// TIA Portal V16 export
// export: Created 2021-11-12T13:31:14.5106173Z, ExportSetting WithDefaults, DisplayName Totally Integrated Automation Portal, DisplayVersion V16 Update 3, DisplayName TIA Portal Version Control Interface, DisplayVersion V16 Update 2, DisplayName TIA Portal Openness, DisplayVersion V16 Update 3, DisplayName SINAMICS Startdrive Advanced, DisplayVersion V16 Update 5, DisplayName SINAMICS Startdrive G130, G150, S120, S150, SINAMICS MV, S210, DisplayVersion V16 Update 5, DisplayName SINAMICS Startdrive G110M, G120, G120C, G120D, G120P, G115D, DisplayVersion V16 Update 5, DisplayName STEP 7 Professional, DisplayVersion V16 Update 3, DisplayName STEP 7 Safety, DisplayVersion V16, DisplayName WinCC UA Professional, DisplayVersion V16 Update 3
FUNCTION_BLOCK "STD_RobotZones"   // FB39, LAD
{ S7_Optimized_Access := 'TRUE' }
VERSION : 0.1
// stored: AutoNumber true, IsIECCheckEnabled false, IsRetainMemResEnabled false, MemoryReserve 100, SetENOAutomatically false, UDAEnableTagReadback false
   VAR_INPUT
      IS_Rob1_ZoneRel : Struct
         Request : Bool;   // Robot requests entering the Station
         Rel : Bool;   // Robot is out of station area
      END_STRUCT;
      IS_Rob2_ZoneRel : Struct
         Request : Bool;   // Robot requests entering the Station
         Rel : Bool;   // Robot is out of station area
      END_STRUCT;
      IS_Rob3_ZoneRel : Struct
         Request : Bool;   // Robot requests entering the Station
         Rel : Bool;   // Robot is out of station area
      END_STRUCT;
      IS_Rob4_ZoneRel : Struct
         Request : Bool;   // Robot requests entering the Station
         Rel : Bool;   // Robot is out of station area
      END_STRUCT;
      IS_Rob5_ZoneRel : Struct
         Request : Bool;   // Robot requests entering the Station
         Rel : Bool;   // Robot is out of station area
      END_STRUCT;
      IS_Rob6_ZoneRel : Struct
         Request : Bool;   // Robot requests entering the Station
         Rel : Bool;   // Robot is out of station area
      END_STRUCT;
      IS_Rob7_ZoneRel : Struct
         Request : Bool;   // Robot requests entering the Station
         Rel : Bool;   // Robot is out of station area
      END_STRUCT;
      IS_Rob8_ZoneRel : Struct
         Request : Bool;   // Robot requests entering the Station
         Rel : Bool;   // Robot is out of station area
      END_STRUCT;
      IB1ZoneRelease : Bool;
   END_VAR
   VAR_OUTPUT
      OS_Rob1_ZoneAll : Struct
         Allowed : Bool;   // Station is allowed for robot entering
      END_STRUCT;
      OS_Rob2_ZoneAll : Struct
         Allowed : Bool;   // Station is allowed for robot entering
      END_STRUCT;
      OS_Rob3_ZoneAll : Struct
         Allowed : Bool;   // Station is allowed for robot entering
      END_STRUCT;
      OS_Rob4_ZoneAll : Struct
         Allowed : Bool;   // Station is allowed for robot entering
      END_STRUCT;
      OS_Rob5_ZoneAll : Struct
         Allowed : Bool;   // Station is allowed for robot entering
      END_STRUCT;
      OS_Rob6_ZoneAll : Struct
         Allowed : Bool;   // Station is allowed for robot entering
      END_STRUCT;
      OS_Rob7_ZoneAll : Struct
         Allowed : Bool;   // Station is allowed for robot entering
      END_STRUCT;
      OS_Rob8_ZoneAll : Struct
         Allowed : Bool;   // Station is allowed for robot entering
      END_STRUCT;
   END_VAR
   VAR_TEMP
      "TB1Zone free" : Bool;
      TS_Rob1_ZoneRel : Struct
         Request : Bool;   // Robot requests entering the Station
         Rel : Bool;   // Robot is out of station area
      END_STRUCT;
      TS_Rob2_ZoneRel : Struct
         Request : Bool;   // Robot requests entering the Station
         Rel : Bool;   // Robot is out of station area
      END_STRUCT;
      TS_Rob3_ZoneRel : Struct
         Request : Bool;   // Robot requests entering the Station
         Rel : Bool;   // Robot is out of station area
      END_STRUCT;
      TS_Rob4_ZoneRel : Struct
         Request : Bool;   // Robot requests entering the Station
         Rel : Bool;   // Robot is out of station area
      END_STRUCT;
      TS_Rob5_ZoneRel : Struct
         Request : Bool;   // Robot requests entering the Station
         Rel : Bool;   // Robot is out of station area
      END_STRUCT;
      TS_Rob6_ZoneRel : Struct
         Request : Bool;   // Robot requests entering the Station
         Rel : Bool;   // Robot is out of station area
      END_STRUCT;
      TS_Rob7_ZoneRel : Struct
         Request : Bool;   // Robot requests entering the Station
         Rel : Bool;   // Robot is out of station area
      END_STRUCT;
      TS_Rob8_ZoneRel : Struct
         Request : Bool;   // Robot requests entering the Station
         Rel : Bool;   // Robot is out of station area
      END_STRUCT;
      TS_Rob1_ZoneAll : Struct
         Allowed : Bool;   // Station is allowed for robot entering
      END_STRUCT;
      TS_Rob2_ZoneAll : Struct
         Allowed : Bool;   // Station is allowed for robot entering
      END_STRUCT;
      TS_Rob3_ZoneAll : Struct
         Allowed : Bool;   // Station is allowed for robot entering
      END_STRUCT;
      TS_Rob4_ZoneAll : Struct
         Allowed : Bool;   // Station is allowed for robot entering
      END_STRUCT;
      TS_Rob5_ZoneAll : Struct
         Allowed : Bool;   // Station is allowed for robot entering
      END_STRUCT;
      TS_Rob6_ZoneAll : Struct
         Allowed : Bool;   // Station is allowed for robot entering
      END_STRUCT;
      TS_Rob7_ZoneAll : Struct
         Allowed : Bool;   // Station is allowed for robot entering
      END_STRUCT;
      TS_Rob8_ZoneAll : Struct
         Allowed : Bool;   // Station is allowed for robot entering
      END_STRUCT;
      TB1ZoneRelease : Bool;
   END_VAR
BEGIN

REGION Network 1: *************** Clear Temporary ***************
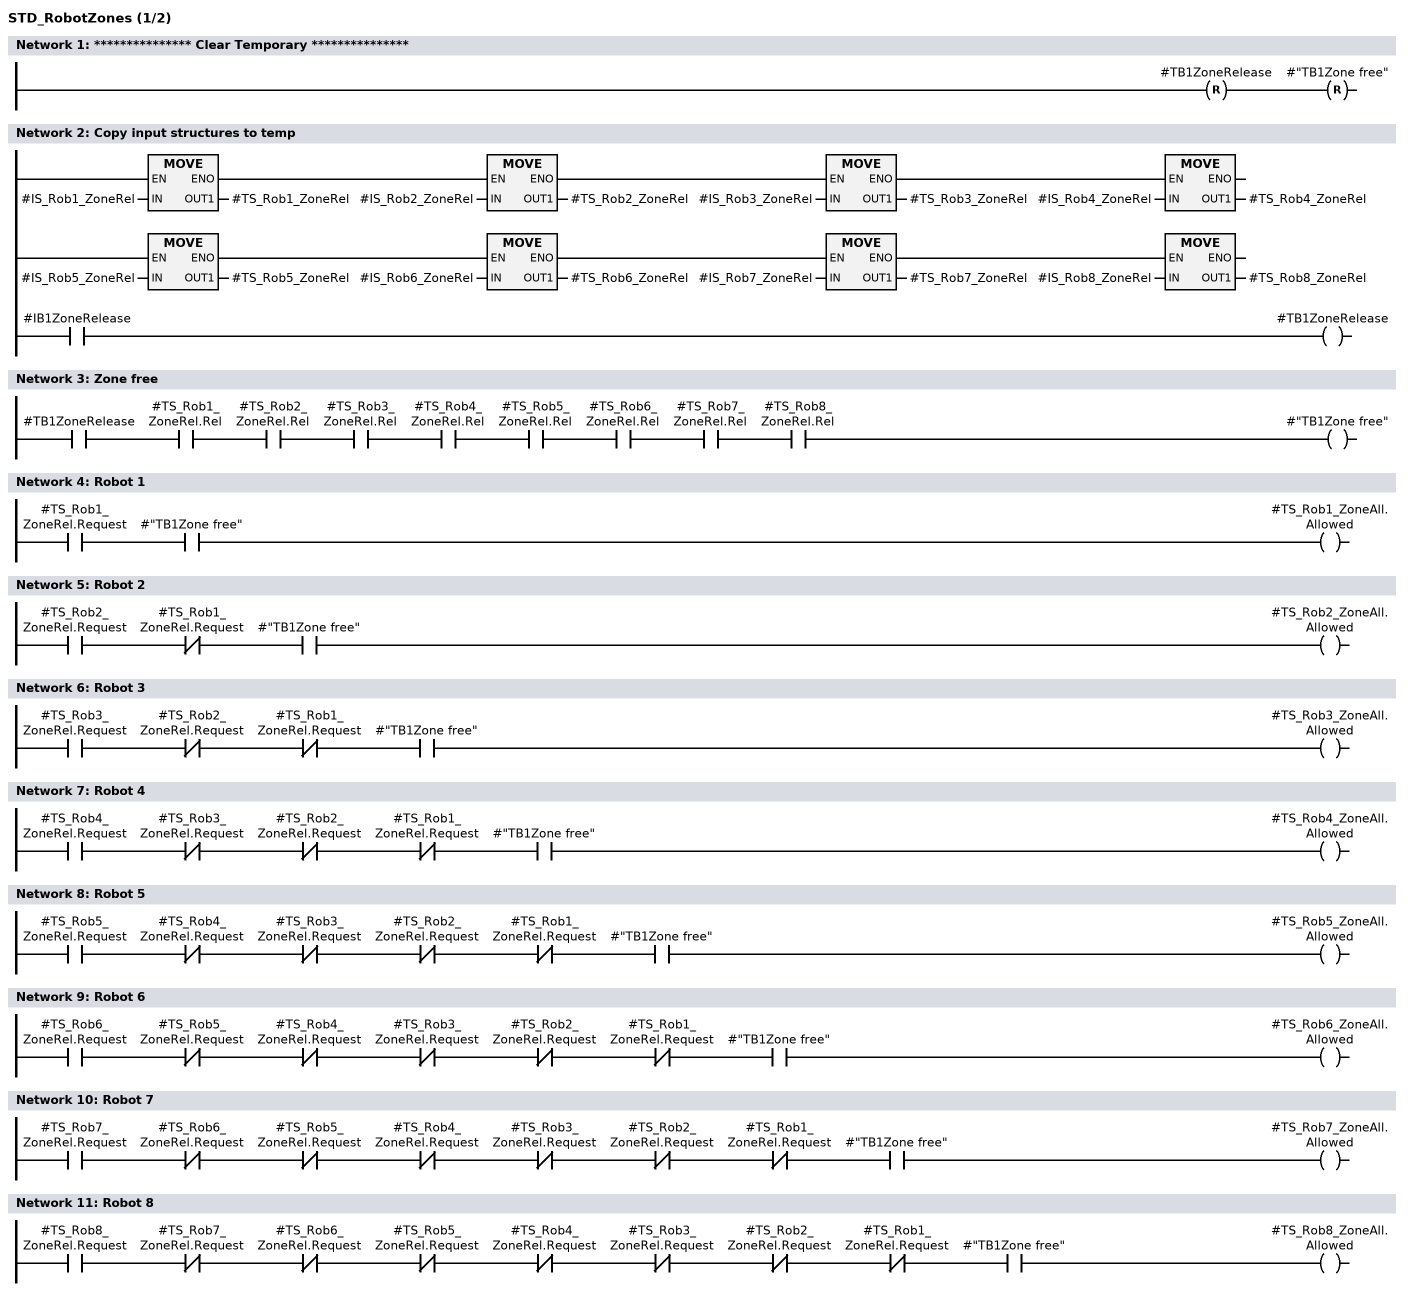
   RUNG wire#powerrail
      R_Coil( #TB1ZoneRelease )
      R_Coil( #"TB1Zone free" )
   END_RUNG
   // the same network as SCL:
   #TB1ZoneRelease := FALSE;
   #"TB1Zone free" := FALSE;
END_REGION

REGION Network 2: Copy input structures to temp
   RUNG wire#powerrail
      Move(in := #IS_Rob1_ZoneRel, out1 => #TS_Rob1_ZoneRel)
      Move(in := #IS_Rob2_ZoneRel, out1 => #TS_Rob2_ZoneRel)
      Move(in := #IS_Rob3_ZoneRel, out1 => #TS_Rob3_ZoneRel)
      Move(in := #IS_Rob4_ZoneRel, out1 => #TS_Rob4_ZoneRel)
   END_RUNG
   RUNG wire#powerrail
      Move(in := #IS_Rob5_ZoneRel, out1 => #TS_Rob5_ZoneRel)
      Move(in := #IS_Rob6_ZoneRel, out1 => #TS_Rob6_ZoneRel)
      Move(in := #IS_Rob7_ZoneRel, out1 => #TS_Rob7_ZoneRel)
      Move(in := #IS_Rob8_ZoneRel, out1 => #TS_Rob8_ZoneRel)
   END_RUNG
   RUNG wire#powerrail
      Contact( #IB1ZoneRelease )
      Coil( #TB1ZoneRelease )
   END_RUNG
   // the same network as SCL:
   #TS_Rob1_ZoneRel := #IS_Rob1_ZoneRel;
   #TS_Rob2_ZoneRel := #IS_Rob2_ZoneRel;
   #TS_Rob3_ZoneRel := #IS_Rob3_ZoneRel;
   #TS_Rob4_ZoneRel := #IS_Rob4_ZoneRel;
   #TS_Rob5_ZoneRel := #IS_Rob5_ZoneRel;
   #TS_Rob6_ZoneRel := #IS_Rob6_ZoneRel;
   #TS_Rob7_ZoneRel := #IS_Rob7_ZoneRel;
   #TS_Rob8_ZoneRel := #IS_Rob8_ZoneRel;
   #TB1ZoneRelease := #IB1ZoneRelease;
END_REGION

REGION Network 3: Zone free
   RUNG wire#powerrail
      Contact( #TB1ZoneRelease )
      Contact( #TS_Rob1_ZoneRel.Rel )
      Contact( #TS_Rob2_ZoneRel.Rel )
      Contact( #TS_Rob3_ZoneRel.Rel )
      Contact( #TS_Rob4_ZoneRel.Rel )
      Contact( #TS_Rob5_ZoneRel.Rel )
      Contact( #TS_Rob6_ZoneRel.Rel )
      Contact( #TS_Rob7_ZoneRel.Rel )
      Contact( #TS_Rob8_ZoneRel.Rel )
      Coil( #"TB1Zone free" )
   END_RUNG
   // the same network as SCL:
   #"TB1Zone free" := #TB1ZoneRelease AND #TS_Rob1_ZoneRel.Rel AND #TS_Rob2_ZoneRel.Rel AND #TS_Rob3_ZoneRel.Rel AND #TS_Rob4_ZoneRel.Rel AND #TS_Rob5_ZoneRel.Rel AND #TS_Rob6_ZoneRel.Rel AND #TS_Rob7_ZoneRel.Rel AND #TS_Rob8_ZoneRel.Rel;
END_REGION

REGION Network 4: Robot 1
   RUNG wire#powerrail
      Contact( #TS_Rob1_ZoneRel.Request )
      Contact( #"TB1Zone free" )
      Coil( #TS_Rob1_ZoneAll.Allowed )
   END_RUNG
   // the same network as SCL:
   #TS_Rob1_ZoneAll.Allowed := #TS_Rob1_ZoneRel.Request AND #"TB1Zone free";
END_REGION

REGION Network 5: Robot 2
   RUNG wire#powerrail
      Contact( #TS_Rob2_ZoneRel.Request )
      I_Contact( #TS_Rob1_ZoneRel.Request )
      Contact( #"TB1Zone free" )
      Coil( #TS_Rob2_ZoneAll.Allowed )
   END_RUNG
   // the same network as SCL:
   #TS_Rob2_ZoneAll.Allowed := #TS_Rob2_ZoneRel.Request AND NOT #TS_Rob1_ZoneRel.Request AND #"TB1Zone free";
END_REGION

REGION Network 6: Robot 3
   RUNG wire#powerrail
      Contact( #TS_Rob3_ZoneRel.Request )
      I_Contact( #TS_Rob2_ZoneRel.Request )
      I_Contact( #TS_Rob1_ZoneRel.Request )
      Contact( #"TB1Zone free" )
      Coil( #TS_Rob3_ZoneAll.Allowed )
   END_RUNG
   // the same network as SCL:
   #TS_Rob3_ZoneAll.Allowed := #TS_Rob3_ZoneRel.Request AND NOT #TS_Rob2_ZoneRel.Request AND NOT #TS_Rob1_ZoneRel.Request AND #"TB1Zone free";
END_REGION

REGION Network 7: Robot 4
   RUNG wire#powerrail
      Contact( #TS_Rob4_ZoneRel.Request )
      I_Contact( #TS_Rob3_ZoneRel.Request )
      I_Contact( #TS_Rob2_ZoneRel.Request )
      I_Contact( #TS_Rob1_ZoneRel.Request )
      Contact( #"TB1Zone free" )
      Coil( #TS_Rob4_ZoneAll.Allowed )
   END_RUNG
   // the same network as SCL:
   #TS_Rob4_ZoneAll.Allowed := #TS_Rob4_ZoneRel.Request AND NOT #TS_Rob3_ZoneRel.Request AND NOT #TS_Rob2_ZoneRel.Request AND NOT #TS_Rob1_ZoneRel.Request AND #"TB1Zone free";
END_REGION

REGION Network 8: Robot 5
   RUNG wire#powerrail
      Contact( #TS_Rob5_ZoneRel.Request )
      I_Contact( #TS_Rob4_ZoneRel.Request )
      I_Contact( #TS_Rob3_ZoneRel.Request )
      I_Contact( #TS_Rob2_ZoneRel.Request )
      I_Contact( #TS_Rob1_ZoneRel.Request )
      Contact( #"TB1Zone free" )
      Coil( #TS_Rob5_ZoneAll.Allowed )
   END_RUNG
   // the same network as SCL:
   #TS_Rob5_ZoneAll.Allowed := #TS_Rob5_ZoneRel.Request AND NOT #TS_Rob4_ZoneRel.Request AND NOT #TS_Rob3_ZoneRel.Request AND NOT #TS_Rob2_ZoneRel.Request AND NOT #TS_Rob1_ZoneRel.Request AND #"TB1Zone free";
END_REGION

REGION Network 9: Robot 6
   RUNG wire#powerrail
      Contact( #TS_Rob6_ZoneRel.Request )
      I_Contact( #TS_Rob5_ZoneRel.Request )
      I_Contact( #TS_Rob4_ZoneRel.Request )
      I_Contact( #TS_Rob3_ZoneRel.Request )
      I_Contact( #TS_Rob2_ZoneRel.Request )
      I_Contact( #TS_Rob1_ZoneRel.Request )
      Contact( #"TB1Zone free" )
      Coil( #TS_Rob6_ZoneAll.Allowed )
   END_RUNG
   // the same network as SCL:
   #TS_Rob6_ZoneAll.Allowed := #TS_Rob6_ZoneRel.Request AND NOT #TS_Rob5_ZoneRel.Request AND NOT #TS_Rob4_ZoneRel.Request AND NOT #TS_Rob3_ZoneRel.Request AND NOT #TS_Rob2_ZoneRel.Request AND NOT #TS_Rob1_ZoneRel.Request AND #"TB1Zone free";
END_REGION

REGION Network 10: Robot 7
   RUNG wire#powerrail
      Contact( #TS_Rob7_ZoneRel.Request )
      I_Contact( #TS_Rob6_ZoneRel.Request )
      I_Contact( #TS_Rob5_ZoneRel.Request )
      I_Contact( #TS_Rob4_ZoneRel.Request )
      I_Contact( #TS_Rob3_ZoneRel.Request )
      I_Contact( #TS_Rob2_ZoneRel.Request )
      I_Contact( #TS_Rob1_ZoneRel.Request )
      Contact( #"TB1Zone free" )
      Coil( #TS_Rob7_ZoneAll.Allowed )
   END_RUNG
   // the same network as SCL:
   #TS_Rob7_ZoneAll.Allowed := #TS_Rob7_ZoneRel.Request AND NOT #TS_Rob6_ZoneRel.Request AND NOT #TS_Rob5_ZoneRel.Request AND NOT #TS_Rob4_ZoneRel.Request AND NOT #TS_Rob3_ZoneRel.Request AND NOT #TS_Rob2_ZoneRel.Request AND NOT #TS_Rob1_ZoneRel.Request AND #"TB1Zone free";
END_REGION

REGION Network 11: Robot 8
   RUNG wire#powerrail
      Contact( #TS_Rob8_ZoneRel.Request )
      I_Contact( #TS_Rob7_ZoneRel.Request )
      I_Contact( #TS_Rob6_ZoneRel.Request )
      I_Contact( #TS_Rob5_ZoneRel.Request )
      I_Contact( #TS_Rob4_ZoneRel.Request )
      I_Contact( #TS_Rob3_ZoneRel.Request )
      I_Contact( #TS_Rob2_ZoneRel.Request )
      I_Contact( #TS_Rob1_ZoneRel.Request )
      Contact( #"TB1Zone free" )
      Coil( #TS_Rob8_ZoneAll.Allowed )
   END_RUNG
   // the same network as SCL:
   #TS_Rob8_ZoneAll.Allowed := #TS_Rob8_ZoneRel.Request AND NOT #TS_Rob7_ZoneRel.Request AND NOT #TS_Rob6_ZoneRel.Request AND NOT #TS_Rob5_ZoneRel.Request AND NOT #TS_Rob4_ZoneRel.Request AND NOT #TS_Rob3_ZoneRel.Request AND NOT #TS_Rob2_ZoneRel.Request AND NOT #TS_Rob1_ZoneRel.Request AND #"TB1Zone free";
END_REGION

REGION Network 12: Copy temp to output structure
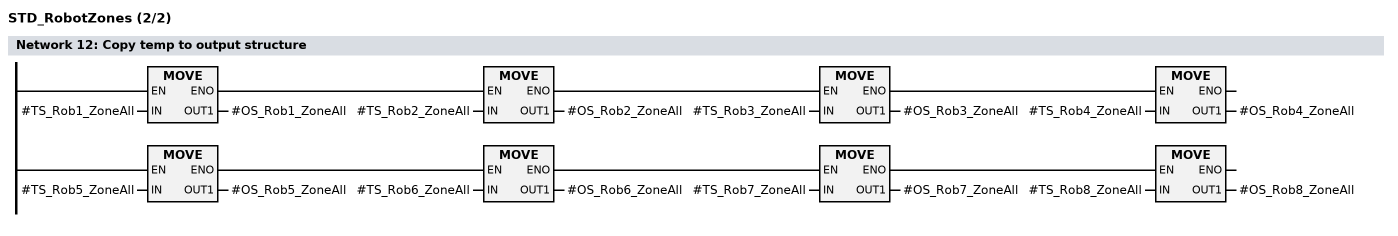
   RUNG wire#powerrail
      Move(in := #TS_Rob1_ZoneAll, out1 => #OS_Rob1_ZoneAll)
      Move(in := #TS_Rob2_ZoneAll, out1 => #OS_Rob2_ZoneAll)
      Move(in := #TS_Rob3_ZoneAll, out1 => #OS_Rob3_ZoneAll)
      Move(in := #TS_Rob4_ZoneAll, out1 => #OS_Rob4_ZoneAll)
   END_RUNG
   RUNG wire#powerrail
      Move(in := #TS_Rob5_ZoneAll, out1 => #OS_Rob5_ZoneAll)
      Move(in := #TS_Rob6_ZoneAll, out1 => #OS_Rob6_ZoneAll)
      Move(in := #TS_Rob7_ZoneAll, out1 => #OS_Rob7_ZoneAll)
      Move(in := #TS_Rob8_ZoneAll, out1 => #OS_Rob8_ZoneAll)
   END_RUNG
   // the same network as SCL:
   #OS_Rob1_ZoneAll := #TS_Rob1_ZoneAll;
   #OS_Rob2_ZoneAll := #TS_Rob2_ZoneAll;
   #OS_Rob3_ZoneAll := #TS_Rob3_ZoneAll;
   #OS_Rob4_ZoneAll := #TS_Rob4_ZoneAll;
   #OS_Rob5_ZoneAll := #TS_Rob5_ZoneAll;
   #OS_Rob6_ZoneAll := #TS_Rob6_ZoneAll;
   #OS_Rob7_ZoneAll := #TS_Rob7_ZoneAll;
   #OS_Rob8_ZoneAll := #TS_Rob8_ZoneAll;
END_REGION
END_FUNCTION_BLOCK
